FUNCTION_BLOCK FB_Drive EXTENDS FB_LinkDataREAL
VAR_INPUT
	nControl  		: BYTE;
	fTargetValue 	: REAL; //Target value to drive
END_VAR

VAR_OUTPUT
	nStatus  		: BYTE;
	fActualValue 	: REAL; //Actual value from drive
END_VAR

SUPER^();
Control := nControl;
ControlData := fTargetValue;
nStatus := Status;
fActualValue := StatusData;

END_FUNCTION_BLOCK

(* stored: Version 1.1.0.1, ProductVersion 3.1.4024.12
   POU FB_Drive: Id {a1a15448-403e-0037-1891-471a9590d7d4}, SpecialFunc None *)
